TYPE ST_Color :
STRUCT
	nTransparency				: BYTE;
	nRed						: BYTE;
	nGreen						: BYTE;
	nBlue						: BYTE;
END_STRUCT
END_TYPE

(* stored: Version 1.1.0.1
   DUT ST_Color: Id {3e36d1c0-4ec6-4a90-b300-adfaa6f6185e} *)
